Staubli VAL3: teachPoints.pgx

program teachPoints()
  local num l_nI
  local num l_nWhich
begin
  //-----------------------------------------------------------------------
  //Header begin
  //Description of program
  //  This program allows you to teach 4 points
  //
  //Traceability
  //  Creation : 07-04-08 - f.Rob
  //Header end
  //-----------------------------------------------------------------------

  userPage()
  cls()
  gotoxy(2,2)
  put(sUsrMess[9+nLangSet])
  gotoxy(1,9)
  put(sUsrMess[13+nLangSet])
  //Function to display navigation keys (F1 through F8) (here F4 with message "Here")
  call usrButtonTxt(4,sUsrMess[26+nLangSet])
  //Loop to remember 4 points
  for l_nI=1 to 4
    gotoxy(2,4)
    //Displays point during the apprenticeship (ex: Teaching of 2.Point)
    putln(sUsrMess[11+nLangSet]+toString("1",l_nI)+sUsrMess[12+nLangSet])
    putln("")
    put("----------------------------------------")
    //Waiting pressing 4 (F4 key) for memorize the point
    wait((get()-270)==4)
    pTempS[l_nI]=here(flange,world)
  endFor
end
